ABB RAPID module: ABSACC.mod

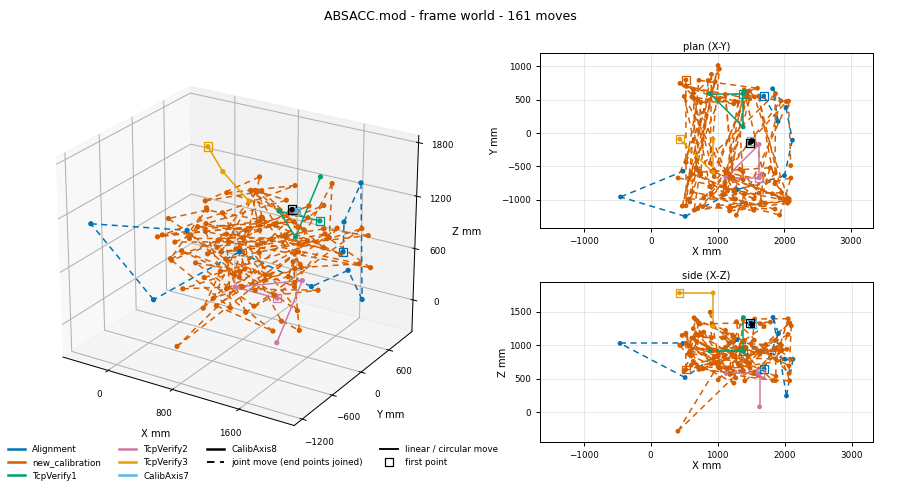
[picture p0: tool path of ABSACC.mod in frame world, 161 of 263 moves have a stored position in this frame; points joined in program order, loops and branches not executed]
%%%
  VERSION:1
  LANGUAGE:ENGLISH
%%%

MODULE ABSACC

    VAR robtarget current_pos   ;
    VAR string log_string;
    VAR iodev file_no;
    VAR num number;
    VAR string outnumber;
    VAR jointtarget jt_current;
    VAR robtarget rt_current;


    VAR num x_pos;
    VAR num y_pos;
    VAR num z_pos;
    VAR num q1_pos;
    VAR num q2_pos;
    VAR num q3_pos;
    VAR num q4_pos;


    VAR jointtarget jpos_after_move;
    VAR jointtarget currentjoints;
    VAR num rob_axis_1;                 ! ????1???
    VAR num rob_axis_2;                 ! ????2???
    VAR num rob_axis_3;                 ! ????3???
    VAR num rob_axis_4;                 ! ????4???
    VAR num rob_axis_5;                 ! ????5???
    VAR num rob_axis_6;                 ! ????6???


CONST robtarget Calib_1:=[[523.49,799.57,640.63],[0.427271,0.615474,0.485528,0.450495],[-1,-1,1,1],[0,9.0000E+09,9.0000E+09,0.000922768,0.0198127,0.000536354]];
CONST robtarget Calib_2:=[[526.56,-1091.2,1181.6],[0.427248,0.615504,0.485478,0.450359],[-1,-1,1,1],[0,9.0000E+09,9.0000E+09,0.000922768,0.020546,0.000486039]];
CONST robtarget Calib_3:=[[720.62,792.84,639.99],[0.427499,0.615430,0.485283,0.450683],[-1,-1,1,1],[0,9.0000E+09,9.0000E+09,0.000922768,0.020546,0.000486039]];
CONST robtarget Calib_4:=[[1598.1,672.95,554.69],[0.427422,0.615259,0.485561,0.450647],[-2,-2,1,1],[0,9.0000E+09,9.0000E+09,0.000922768,0.0181016,0.000506165]];
CONST robtarget Calib_5:=[[1022.6,515.85,667.24],[0.427491,0.615409,0.485531,0.450370],[-2,-2,1,1],[0,9.0000E+09,9.0000E+09,0.000922768,0.0181016,0.000506165]];
CONST robtarget Calib_6:=[[573.72,-670.12,994.4],[0.427363,0.615467,0.485428,0.450324],[-1,-2,2,1],[0,9.0000E+09,9.0000E+09,0.000770224,0.0198127,0.000536354]];
CONST robtarget Calib_7:=[[723.98,-576.9,1336.5],[0.427491,0.615540,0.485574,0.450598],[-2,-2,1,1],[0,9.0000E+09,9.0000E+09,0.000922768,0.0181016,0.000506165]];
CONST robtarget Calib_8:=[[582.16,-1033.6,910.76],[0.427404,0.615425,0.485431,0.450648],[-1,-2,2,1],[0,9.0000E+09,9.0000E+09,0.000770224,0.0198127,0.000536354]];
CONST robtarget Calib_9:=[[1006.3,1014.5,850.46],[0.427169,0.615279,0.485385,0.450491],[-1,-1,1,1],[0,9.0000E+09,9.0000E+09,0.000922768,0.0198127,0.000536354]];
CONST robtarget Calib_10:=[[566.63,-990.26,872.37],[0.427234,0.615354,0.485638,0.450740],[-1,-1,1,1],[0,9.0000E+09,9.0000E+09,0.000922768,0.0198127,0.000536354]];
CONST robtarget Calib_11:=[[1269.8,-989.4,513.75],[0.427266,0.615492,0.485274,0.450510],[-1,-1,1,1],[0,9.0000E+09,9.0000E+09,0.000922768,0.020546,0.000486039]];
CONST robtarget Calib_12:=[[1116.4,-816.34,1225.6],[0.427348,0.615327,0.485558,0.450713],[-2,-2,1,1],[0,9.0000E+09,9.0000E+09,0.000922768,0.0181016,0.000506165]];
CONST robtarget Calib_13:=[[1482.7,514.18,659.18],[0.427130,0.615463,0.485370,0.450503],[-1,-2,2,1],[0,9.0000E+09,9.0000E+09,0.000770224,0.0198127,0.000536354]];
CONST robtarget Calib_14:=[[531.86,699.88,1033.4],[0.427259,0.615357,0.485446,0.450699],[-1,-1,1,1],[0,9.0000E+09,9.0000E+09,0.000922768,0.020546,0.000486039]];
CONST robtarget Calib_15:=[[635.74,656.93,761.23],[0.427346,0.615523,0.485389,0.450649],[-1,-1,1,1],[0,9.0000E+09,9.0000E+09,0.000922768,0.020546,0.000486039]];
CONST robtarget Calib_16:=[[1241.2,439.93,437],[0.427180,0.615539,0.485346,0.450641],[-2,-2,1,1],[0,9.0000E+09,9.0000E+09,0.000922768,0.0181016,0.000506165]];
CONST robtarget Calib_17:=[[612.86,545.6,1108.6],[0.427352,0.615273,0.485557,0.450373],[-2,-2,1,1],[0,9.0000E+09,9.0000E+09,0.000922768,0.0181016,0.000506165]];
CONST robtarget Calib_18:=[[856.4,789.38,964.12],[0.427443,0.615400,0.485449,0.450538],[-1,-1,1,1],[0,9.0000E+09,9.0000E+09,0.000922768,0.0198127,0.000536354]];
CONST robtarget Calib_19:=[[746.48,-623.31,1183.2],[0.427151,0.615444,0.485503,0.450550],[-1,-1,1,1],[0,9.0000E+09,9.0000E+09,0.000922768,0.0198127,0.000536354]];
CONST robtarget Calib_20:=[[498.99,549.58,619.65],[0.427533,0.615524,0.485442,0.450402],[-1,-1,1,1],[0,9.0000E+09,9.0000E+09,0.000922768,0.0198127,0.000536354]];
CONST robtarget Calib_21:=[[1260.9,-903.01,847.24],[0.427221,0.615530,0.485537,0.450347],[-1,-1,1,1],[0,9.0000E+09,9.0000E+09,0.000922768,0.0198127,0.000536354]];
CONST robtarget Calib_22:=[[1115.2,580.02,967.53],[0.427294,0.615266,0.485509,0.450741],[-1,-2,2,1],[0,9.0000E+09,9.0000E+09,0.000770224,0.0198127,0.000536354]];
CONST robtarget Calib_23:=[[1222.6,-669.28,1154.2],[0.427349,0.615383,0.485339,0.450300],[-1,-1,1,1],[0,9.0000E+09,9.0000E+09,0.000922768,0.0198127,0.000536354]];
CONST robtarget Calib_24:=[[1384,-699.69,623.11],[0.427265,0.615494,0.485307,0.450350],[-1,-1,1,1],[0,9.0000E+09,9.0000E+09,0.000922768,0.020546,0.000486039]];
CONST robtarget Calib_25:=[[1308.7,467.72,716.41],[0.427497,0.615508,0.485570,0.450737],[-1,-2,2,1],[0,9.0000E+09,9.0000E+09,0.000770224,0.0198127,0.000536354]];
CONST robtarget Calib_26:=[[1108.9,-758.92,1117],[0.427089,0.615547,0.485259,0.450374],[-2,-2,1,1],[0,9.0000E+09,9.0000E+09,0.000922768,0.0181016,0.000506165]];
CONST robtarget Calib_27:=[[701,-1126.7,1157],[0.427424,0.615529,0.485327,0.450564],[-1,-2,2,1],[0,9.0000E+09,9.0000E+09,0.000770224,0.0198127,0.000536354]];
CONST robtarget Calib_28:=[[792.13,-971.51,1198.2],[0.427131,0.615367,0.485491,0.450773],[-2,-2,1,1],[0,9.0000E+09,9.0000E+09,0.000922768,0.0181016,0.000506165]];
CONST robtarget Calib_29:=[[1126,-591.56,665.82],[0.427307,0.615501,0.485324,0.450344],[-1,-1,1,1],[0,9.0000E+09,9.0000E+09,0.000922768,0.020546,0.000486039]];
CONST robtarget Calib_30:=[[635.98,600.07,1249.9],[0.427092,0.615395,0.485545,0.450727],[-1,-1,1,1],[0,9.0000E+09,9.0000E+09,0.000922768,0.0198127,0.000536354]];
CONST robtarget Calib_31:=[[674,-522.19,1382.2],[0.427363,0.615521,0.485308,0.450727],[-1,-2,2,1],[0,9.0000E+09,9.0000E+09,0.000770224,0.0198127,0.000536354]];
CONST robtarget Calib_32:=[[748.13,462.02,1157.5],[0.427338,0.615483,0.485637,0.450429],[-1,-2,2,1],[0,9.0000E+09,9.0000E+09,0.000770224,0.0198127,0.000536354]];
CONST robtarget Calib_33:=[[1259.1,477.91,827.2],[0.427346,0.615281,0.485321,0.450436],[-1,-2,2,1],[0,9.0000E+09,9.0000E+09,0.000770224,0.0198127,0.000536354]];
CONST robtarget Calib_34:=[[435.05,747.18,1000.2],[0.427446,0.615477,0.485492,0.450579],[-2,-2,1,1],[0,9.0000E+09,9.0000E+09,0.000922768,0.0181016,0.000506165]];
CONST robtarget Calib_35:=[[700.02,500.97,685.14],[0.427265,0.615499,0.485337,0.450378],[-1,-1,1,1],[0,9.0000E+09,9.0000E+09,0.000922768,0.0198127,0.000536354]];
CONST robtarget Calib_36:=[[527.77,-439.15,1030.3],[0.427281,0.615357,0.485288,0.450618],[-1,-1,1,1],[0,9.0000E+09,9.0000E+09,0.000922768,0.0198127,0.000536354]];
CONST robtarget Calib_37:=[[964.85,768.97,744],[0.427293,0.615355,0.485428,0.450593],[-2,-2,1,1],[0,9.0000E+09,9.0000E+09,0.000922768,0.0181016,0.000506165]];
CONST robtarget Calib_38:=[[469.94,-1095.9,1149],[0.427187,0.615553,0.485531,0.450739],[-1,-1,1,1],[0,9.0000E+09,9.0000E+09,0.000922768,0.0198127,0.000536354]];
CONST robtarget Calib_39:=[[908.06,882.12,1111.7],[0.427135,0.615427,0.485420,0.450717],[-2,-2,1,1],[0,9.0000E+09,9.0000E+09,0.000922768,0.0181016,0.000506165]];
CONST robtarget Calib_40:=[[889.34,-450.25,1494.7],[0.427395,0.615312,0.485584,0.450720],[-2,-2,1,1],[0,9.0000E+09,9.0000E+09,0.000922768,0.0181016,0.000506165]];
CONST robtarget Calib_41:=[[1026.6,961.76,736],[0.427363,0.615234,0.485457,0.450402],[-1,-1,1,1],[0,9.0000E+09,9.0000E+09,0.000922768,0.020546,0.000486039]];
CONST robtarget Calib_42:=[[406.52,-673.62,-280.36],[0.427280,0.615259,0.485296,0.450679],[-1,-1,1,1],[0,9.0000E+09,9.0000E+09,0.000922768,0.020546,0.000486039]];
CONST robtarget Calib_43:=[[2074.8,-1023.6,1336],[0.337031,0.670436,0.287182,0.595360],[-1,-1,1,1],[9.0000E+09,9.0000E+09,9.0000E+09,9.0000E+09,9.0000E+09,9.0000E+09]];
CONST robtarget Calib_44:=[[1181.5,-1112.6,566.66],[0.337038,0.670376,0.287151,0.595390],[-1,-1,2,1],[9.0000E+09,9.0000E+09,9.0000E+09,9.0000E+09,9.0000E+09,9.0000E+09]];
CONST robtarget Calib_45:=[[1861.9,-1141,473.33],[0.337097,0.670438,0.287154,0.595390],[-1,0,1,1],[9.0000E+09,9.0000E+09,9.0000E+09,9.0000E+09,9.0000E+09,9.0000E+09]];
CONST robtarget Calib_46:=[[901.25,-902.02,725.94],[0.337013,0.670422,0.287231,0.595328],[-1,-1,1,1],[9.0000E+09,9.0000E+09,9.0000E+09,9.0000E+09,9.0000E+09,9.0000E+09]];
CONST robtarget Calib_47:=[[1948.9,483.67,997.95],[0.337045,0.670418,0.287223,0.595385],[-1,-1,1,1],[9.0000E+09,9.0000E+09,9.0000E+09,9.0000E+09,9.0000E+09,9.0000E+09]];
CONST robtarget Calib_48:=[[1546.2,-986.65,603.41],[0.337073,0.670424,0.287150,0.595345],[0,0,1,1],[9.0000E+09,9.0000E+09,9.0000E+09,9.0000E+09,9.0000E+09,9.0000E+09]];
CONST robtarget Calib_49:=[[605.19,-604.49,704.07],[0.337059,0.670417,0.287152,0.595308],[0,0,1,1],[9.0000E+09,9.0000E+09,9.0000E+09,9.0000E+09,9.0000E+09,9.0000E+09]];
CONST robtarget Calib_50:=[[1718.7,-1051.7,1013.8],[0.337045,0.670449,0.287202,0.595417],[0,0,0,1],[9.0000E+09,9.0000E+09,9.0000E+09,9.0000E+09,9.0000E+09,9.0000E+09]];
CONST robtarget Calib_51:=[[1182.6,-676.82,1033.8],[0.337024,0.670403,0.287174,0.595407],[-1,-1,2,1],[9.0000E+09,9.0000E+09,9.0000E+09,9.0000E+09,9.0000E+09,9.0000E+09]];
CONST robtarget Calib_52:=[[1545.3,-1159,1076.6],[0.337084,0.670398,0.287161,0.595421],[0,0,1,1],[9.0000E+09,9.0000E+09,9.0000E+09,9.0000E+09,9.0000E+09,9.0000E+09]];
CONST robtarget Calib_53:=[[774.81,-1104.3,649.63],[0.337065,0.670394,0.287225,0.595345],[0,1,0,1],[9.0000E+09,9.0000E+09,9.0000E+09,9.0000E+09,9.0000E+09,9.0000E+09]];
CONST robtarget Calib_54:=[[1176.9,-617.93,582.71],[0.337054,0.670449,0.287235,0.595440],[0,0,0,1],[9.0000E+09,9.0000E+09,9.0000E+09,9.0000E+09,9.0000E+09,9.0000E+09]];
CONST robtarget Calib_55:=[[1933.5,-974.06,1016],[0.337054,0.670455,0.287213,0.595317],[-1,-1,1,1],[9.0000E+09,9.0000E+09,9.0000E+09,9.0000E+09,9.0000E+09,9.0000E+09]];
CONST robtarget Calib_56:=[[2052.5,-974.74,1397.5],[0.337096,0.670387,0.287178,0.595388],[0,0,1,1],[9.0000E+09,9.0000E+09,9.0000E+09,9.0000E+09,9.0000E+09,9.0000E+09]];
CONST robtarget Calib_57:=[[1552.8,542.67,1393.9],[0.337078,0.670388,0.287224,0.595338],[0,0,1,1],[9.0000E+09,9.0000E+09,9.0000E+09,9.0000E+09,9.0000E+09,9.0000E+09]];
CONST robtarget Calib_58:=[[1479.6,633.54,729.48],[0.337077,0.670453,0.287230,0.595399],[-1,-1,1,1],[9.0000E+09,9.0000E+09,9.0000E+09,9.0000E+09,9.0000E+09,9.0000E+09]];
CONST robtarget Calib_59:=[[942.08,-556.73,811.34],[0.337051,0.670394,0.287182,0.595426],[0,0,1,1],[9.0000E+09,9.0000E+09,9.0000E+09,9.0000E+09,9.0000E+09,9.0000E+09]];
CONST robtarget Calib_60:=[[1865.4,-737.13,799.35],[0.337079,0.670347,0.287195,0.595413],[0,0,1,1],[9.0000E+09,9.0000E+09,9.0000E+09,9.0000E+09,9.0000E+09,9.0000E+09]];
CONST robtarget Calib_61:=[[2050.6,-1051.8,1162.8],[0.337039,0.670451,0.287233,0.595373],[-1,-1,2,1],[9.0000E+09,9.0000E+09,9.0000E+09,9.0000E+09,9.0000E+09,9.0000E+09]];
CONST robtarget Calib_62:=[[1179.9,-1167.8,668.09],[0.337018,0.670357,0.287230,0.595352],[0,0,1,1],[9.0000E+09,9.0000E+09,9.0000E+09,9.0000E+09,9.0000E+09,9.0000E+09]];
CONST robtarget Calib_63:=[[1250.1,-852.23,1106.8],[0.337032,0.670393,0.287200,0.595412],[0,0,1,1],[9.0000E+09,9.0000E+09,9.0000E+09,9.0000E+09,9.0000E+09,9.0000E+09]];
CONST robtarget Calib_64:=[[1380.7,-581.78,1383.3],[0.337027,0.670421,0.287218,0.595331],[-2,-2,2,1],[9.0000E+09,9.0000E+09,9.0000E+09,9.0000E+09,9.0000E+09,9.0000E+09]];
CONST robtarget Calib_65:=[[1335.1,-543.79,968.31],[0.337051,0.670354,0.287205,0.595374],[0,1,0,1],[9.0000E+09,9.0000E+09,9.0000E+09,9.0000E+09,9.0000E+09,9.0000E+09]];
CONST robtarget Calib_66:=[[1622.8,-900.39,876.91],[0.337041,0.670454,0.287187,0.595438],[0,0,0,1],[9.0000E+09,9.0000E+09,9.0000E+09,9.0000E+09,9.0000E+09,9.0000E+09]];
CONST robtarget Calib_67:=[[1861.8,-601.93,954.03],[0.337062,0.670370,0.287184,0.595412],[-1,-1,2,1],[9.0000E+09,9.0000E+09,9.0000E+09,9.0000E+09,9.0000E+09,9.0000E+09]];
CONST robtarget Calib_68:=[[1869.1,592.3,538],[0.337015,0.670426,0.287199,0.595320],[0,0,1,1],[9.0000E+09,9.0000E+09,9.0000E+09,9.0000E+09,9.0000E+09,9.0000E+09]];
CONST robtarget Calib_69:=[[692.16,-548.27,1056.3],[0.337058,0.670360,0.287213,0.595396],[-2,-2,2,1],[9.0000E+09,9.0000E+09,9.0000E+09,9.0000E+09,9.0000E+09,9.0000E+09]];
CONST robtarget Calib_70:=[[1101.7,-909.92,848.42],[0.337048,0.670416,0.287158,0.595327],[-1,-1,2,1],[9.0000E+09,9.0000E+09,9.0000E+09,9.0000E+09,9.0000E+09,9.0000E+09]];
CONST robtarget Calib_71:=[[1007.8,-1088,485.37],[0.337071,0.670388,0.287186,0.595329],[0,1,0,1],[9.0000E+09,9.0000E+09,9.0000E+09,9.0000E+09,9.0000E+09,9.0000E+09]];
CONST robtarget Calib_72:=[[1421.7,-1049.4,969.62],[0.337024,0.670400,0.287209,0.595388],[-2,-2,2,1],[9.0000E+09,9.0000E+09,9.0000E+09,9.0000E+09,9.0000E+09,9.0000E+09]];
CONST robtarget Calib_73:=[[617.49,-882.09,948.54],[0.337019,0.670425,0.287148,0.595386],[-1,-1,1,1],[9.0000E+09,9.0000E+09,9.0000E+09,9.0000E+09,9.0000E+09,9.0000E+09]];
CONST robtarget Calib_74:=[[1931.9,-1230.9,917.13],[0.337103,0.670350,0.287183,0.595318],[0,1,0,1],[9.0000E+09,9.0000E+09,9.0000E+09,9.0000E+09,9.0000E+09,9.0000E+09]];
CONST robtarget Calib_75:=[[2100.7,-673.62,791.58],[0.337065,0.670443,0.287160,0.595345],[-1,0,1,1],[9.0000E+09,9.0000E+09,9.0000E+09,9.0000E+09,9.0000E+09,9.0000E+09]];
CONST robtarget Calib_76:=[[1149.7,-869.76,649.62],[0.337094,0.670428,0.287147,0.595325],[-1,0,1,1],[9.0000E+09,9.0000E+09,9.0000E+09,9.0000E+09,9.0000E+09,9.0000E+09]];
CONST robtarget Calib_77:=[[1431.9,625.97,764.27],[0.337014,0.670388,0.287161,0.595331],[-1,-1,2,1],[9.0000E+09,9.0000E+09,9.0000E+09,9.0000E+09,9.0000E+09,9.0000E+09]];
CONST robtarget Calib_78:=[[949.02,-653.32,926.53],[0.337059,0.670433,0.287179,0.595404],[-1,0,1,1],[9.0000E+09,9.0000E+09,9.0000E+09,9.0000E+09,9.0000E+09,9.0000E+09]];
CONST robtarget Calib_79:=[[640.82,524,1107.8],[0.337046,0.670413,0.287183,0.595344],[-1,-1,2,1],[9.0000E+09,9.0000E+09,9.0000E+09,9.0000E+09,9.0000E+09,9.0000E+09]];
CONST robtarget Calib_80:=[[881.01,-803.61,947.89],[0.337084,0.670403,0.287189,0.595343],[0,1,0,1],[9.0000E+09,9.0000E+09,9.0000E+09,9.0000E+09,9.0000E+09,9.0000E+09]];
CONST robtarget Calib_81:=[[2031.7,473.01,942.05],[0.337084,0.670381,0.287185,0.595336],[0,0,1,1],[9.0000E+09,9.0000E+09,9.0000E+09,9.0000E+09,9.0000E+09,9.0000E+09]];
CONST robtarget Calib_82:=[[1448.7,566.46,849.39],[0.337036,0.670409,0.287180,0.595326],[0,0,1,1],[9.0000E+09,9.0000E+09,9.0000E+09,9.0000E+09,9.0000E+09,9.0000E+09]];
CONST robtarget Calib_83:=[[1072.2,-924.1,1112.3],[0.337049,0.670411,0.287235,0.595327],[0,0,0,1],[9.0000E+09,9.0000E+09,9.0000E+09,9.0000E+09,9.0000E+09,9.0000E+09]];
CONST robtarget Calib_84:=[[1398.2,648.97,1074.8],[0.337050,0.670360,0.287199,0.595382],[-1,-1,1,1],[9.0000E+09,9.0000E+09,9.0000E+09,9.0000E+09,9.0000E+09,9.0000E+09]];
CONST robtarget Calib_85:=[[1692.1,-629.73,1280.4],[0.337086,0.670389,0.287196,0.595338],[-2,-2,2,1],[9.0000E+09,9.0000E+09,9.0000E+09,9.0000E+09,9.0000E+09,9.0000E+09]];
CONST robtarget Calib_86:=[[1635.2,-1070.1,1324.1],[0.337011,0.670430,0.287237,0.595376],[-1,-1,2,1],[9.0000E+09,9.0000E+09,9.0000E+09,9.0000E+09,9.0000E+09,9.0000E+09]];
CONST robtarget Calib_87:=[[1787,-520.57,1346.8],[0.337047,0.670444,0.287202,0.595388],[-1,-1,2,1],[9.0000E+09,9.0000E+09,9.0000E+09,9.0000E+09,9.0000E+09,9.0000E+09]];
CONST robtarget Calib_88:=[[735.47,-585.55,1318.4],[0.337086,0.670436,0.287148,0.595336],[-2,-2,2,1],[9.0000E+09,9.0000E+09,9.0000E+09,9.0000E+09,9.0000E+09,9.0000E+09]];
CONST robtarget Calib_89:=[[647.3,-1156,1412],[0.337021,0.670442,0.287213,0.595341],[-1,-1,2,1],[9.0000E+09,9.0000E+09,9.0000E+09,9.0000E+09,9.0000E+09,9.0000E+09]];
CONST robtarget Calib_90:=[[2064.3,-1013.5,695.66],[0.337032,0.670388,0.287233,0.595308],[0,0,0,1],[9.0000E+09,9.0000E+09,9.0000E+09,9.0000E+09,9.0000E+09,9.0000E+09]];
CONST robtarget Calib_91:=[[914.78,-574.42,1323.8],[0.337011,0.670425,0.287187,0.595439],[-1,-1,2,1],[9.0000E+09,9.0000E+09,9.0000E+09,9.0000E+09,9.0000E+09,9.0000E+09]];
CONST robtarget Calib_92:=[[1822.4,-911.38,476.82],[0.337067,0.670456,0.287225,0.595396],[-1,-1,1,1],[9.0000E+09,9.0000E+09,9.0000E+09,9.0000E+09,9.0000E+09,9.0000E+09]];
CONST robtarget Calib_93:=[[2074.2,-987.78,472.31],[0.337079,0.670363,0.287184,0.595396],[-1,-1,2,1],[9.0000E+09,9.0000E+09,9.0000E+09,9.0000E+09,9.0000E+09,9.0000E+09]];
CONST robtarget Calib_94:=[[1860.3,-759.59,1077.8],[0.337047,0.670419,0.287236,0.595422],[-2,-2,2,1],[9.0000E+09,9.0000E+09,9.0000E+09,9.0000E+09,9.0000E+09,9.0000E+09]];
CONST robtarget Calib_95:=[[1614.9,555.68,899.4],[0.337047,0.670434,0.287180,0.595372],[0,0,0,1],[9.0000E+09,9.0000E+09,9.0000E+09,9.0000E+09,9.0000E+09,9.0000E+09]];
CONST robtarget Calib_96:=[[1960.6,-894.35,930.39],[0.337070,0.670442,0.287225,0.595321],[-1,-1,2,1],[9.0000E+09,9.0000E+09,9.0000E+09,9.0000E+09,9.0000E+09,9.0000E+09]];
CONST robtarget Calib_97:=[[1405.1,-914.47,469.92],[0.337108,0.670454,0.287208,0.595360],[0,1,0,1],[9.0000E+09,9.0000E+09,9.0000E+09,9.0000E+09,9.0000E+09,9.0000E+09]];
CONST robtarget Calib_98:=[[1281,-1232.4,1353.2],[0.337026,0.670376,0.287182,0.595400],[-2,-2,2,1],[9.0000E+09,9.0000E+09,9.0000E+09,9.0000E+09,9.0000E+09,9.0000E+09]];
CONST robtarget Calib_99:=[[2064.8,479.5,583.13],[0.337055,0.670394,0.287212,0.595368],[0,0,1,1],[9.0000E+09,9.0000E+09,9.0000E+09,9.0000E+09,9.0000E+09,9.0000E+09]];
CONST robtarget Calib_100:=[[2097.5,-487.03,1291.9],[0.337063,0.670458,0.287190,0.595322],[-1,-1,2,1],[9.0000E+09,9.0000E+09,9.0000E+09,9.0000E+09,9.0000E+09,9.0000E+09]];







CONST jointtarget JT_Set1_1:=[[53.1735,26.9510,23.3573,73.4890,-59.9300,59.2650],[0,9000000000.0,9000000000.0,0,0,0]];
CONST jointtarget JT_Set1_2:=[[104.8875,-39.2172,32.0501,101.4420,-111.1420,5.5760],[0,9000000000.0,9000000000.0,0,0,0]];
CONST jointtarget JT_Set1_3:=[[-0.5260,-0.9171,-22.1124,172.3270,-36.5000,-74.4910],[0,9000000000.0,9000000000.0,0,0,0]];
CONST jointtarget JT_Set1_4:=[[-71.4352,25.7651,25.2310,-79.7280,-64.8550,137.7380],[0,9000000000.0,9000000000.0,0,0,0]];
CONST jointtarget JT_Set1_5:=[[-33.2693,73.5127,6.3150,-29.5740,-67.8700,103.3770],[0,9000000000.0,9000000000.0,0,0,0]];
CONST jointtarget JT_Set1_6:=[[-10.4906,14.7639,-6.2399,-133.2560,-7.0380,230.5130],[0,9000000000.0,9000000000.0,0,0,0]];
CONST jointtarget JT_Set1_7:=[[-93.3527,9.8440,13.8280,-101.4370,-83.0510,165.4770],[0,9000000000.0,9000000000.0,0,0,0]];
CONST jointtarget JT_Set1_8:=[[11.7457,37.5557,36.3356,18.9030,-61.4260,92.9380],[0,9000000000.0,9000000000.0,0,0,0]];
CONST jointtarget JT_Set1_9:=[[21.7410,14.7129,-20.7875,125.9430,-33.0750,-25.9510],[0,9000000000.0,9000000000.0,0,0,0]];
CONST jointtarget JT_Set1_10:=[[-2.9191,4.9374,-1.3727,167.2410,-9.9250,-68.6510],[0,9000000000.0,9000000000.0,0,0,0]];
CONST jointtarget JT_Set1_11:=[[-5.6872,43.8374,27.8881,-61.6498,-69.5127,61.2],[0,9000000000.0,9000000000.0,0,0,0]];
CONST jointtarget JT_Set1_12:=[[50.3079,41.8227,-20.4018,120.7182,-152.8732,-46.8],[0,9000000000.0,9000000000.0,0,0,0]];
CONST jointtarget JT_Set1_13:=[[84.3385,18.9432,34.5532,160.8424,-29.5414,-118.8],[0,9000000000.0,9000000000.0,0,0,0]];
CONST jointtarget JT_Set1_14:=[[58.297,-2.0746,27.5285,-154.2974,-61.9657,-72.0],[0,9000000000.0,9000000000.0,0,0,0]];
CONST jointtarget JT_Set1_15:=[[32.8735,-30.4364,-59.6442,95.92,-47.9329,-86.4],[0,9000000000.0,9000000000.0,0,0,0]];
CONST jointtarget JT_Set1_16:=[[-33.6427,-18.5643,-12.0604,48.1328,-64.5324,126.0],[0,9000000000.0,9000000000.0,0,0,0]];
CONST jointtarget JT_Set1_17:=[[70.3802,17.2132,-4.0173,-21.5256,-130.5416,43.2],[0,9000000000.0,9000000000.0,0,0,0]];
CONST jointtarget JT_Set1_18:=[[89.0267,-51.2569,56.4018,-36.8517,-171.8904,-39.6],[0,9000000000.0,9000000000.0,0,0,0]];
CONST jointtarget JT_Set1_19:=[[5.7192,-2.5391,54.5482,-94.111,-150.4586,75.6],[0,9000000000.0,9000000000.0,0,0,0]];
CONST jointtarget JT_Set1_20:=[[-0.2027,50.2882,-24.7763,71.1219,-88.2809,97.2],[0,9000000000.0,9000000000.0,0,0,0]];
CONST jointtarget JT_Set1_21:=[[40.4823,-51.699,50.7331,136.0443,-70.7312,162.0],[0,9000000000.0,9000000000.0,0,0,0]];
CONST jointtarget JT_Set1_22:=[[-80.423,25.9753,1.6904,-171.4325,-135.2349,-75.6],[0,9000000000.0,9000000000.0,0,0,0]];
CONST jointtarget JT_Set1_23:=[[11.1889,-11.9535,-14.0107,-141.8983,-94.014,108.0],[0,9000000000.0,9000000000.0,0,0,0]];
CONST jointtarget JT_Set1_24:=[[54.1566,23.8297,-25.9466,8.0085,-89.427,165.6],[0,9000000000.0,9000000000.0,0,0,0]];
CONST jointtarget JT_Set1_25:=[[-59.19,39.8806,42.4357,-114.1731,-100.9528,-97.2],[0,9000000000.0,9000000000.0,0,0,0]];
CONST jointtarget JT_Set1_26:=[[22.8731,-54.4881,33.5123,-146.6343,-111.7156,-28.8],[0,9000000000.0,9000000000.0,0,0,0]];
CONST jointtarget JT_Set1_27:=[[-17.9117,51.6859,-47.3684,-76.9759,-37.8145,-50.4],[0,9000000000.0,9000000000.0,0,0,0]];
CONST jointtarget JT_Set1_28:=[[66.8969,-54.1454,-30.6363,156.1064,-124.7502,7.2],[0,9000000000.0,9000000000.0,0,0,0]];
CONST jointtarget JT_Set1_29:=[[27.4745,30.9191,-59.737,55.7958,-158.4348,28.8],[0,9000000000.0,9000000000.0,0,0,0]];
CONST jointtarget JT_Set1_30:=[[-14.9131,37.7906,30.1398,75.8579,-55.2498,21.6],[0,9000000000.0,9000000000.0,0,0,0]];
CONST jointtarget JT_Set1_31:=[[3.0179,52.3778,-47.9993,-78.7849,-44.7651,-140.4],[0,9000000000.0,9000000000.0,0,0,0]];
CONST jointtarget JT_Set1_32:=[[-83.9819,-55.1498,-7.8347,108.3191,-115.4676,79.2],[0,9000000000.0,9000000000.0,0,0,0]];
CONST jointtarget JT_Set1_33:=[[25.0821,42.0558,5.111,-1.4635,-85.986,-115.2],[0,9000000000.0,9000000000.0,0,0,0]];
CONST jointtarget JT_Set1_34:=[[76.0705,-26.6255,7.5352,30.9977,-14.0699,-111.6],[0,9000000000.0,9000000000.0,0,0,0]];
CONST jointtarget JT_Set1_35:=[[19.3661,-58.9602,39.5929,-86.448,-116.7437,-10.8],[0,9000000000.0,9000000000.0,0,0,0]];
CONST jointtarget JT_Set1_36:=[[80.2267,36.5199,-43.3022,143.7073,-46.3699,57.6],[0,9000000000.0,9000000000.0,0,0,0]];
CONST jointtarget JT_Set1_37:=[[48.0395,-22.389,-23.9848,-24.4526,-136.8864,-68.4],[0,9000000000.0,9000000000.0,0,0,0]];
CONST jointtarget JT_Set1_38:=[[18.7521,-39.7648,-9.1071,80.5939,-43.1136,-169.2],[0,9000000000.0,9000000000.0,0,0,0]];
CONST jointtarget JT_Set1_39:=[[-19.8231,-9.8027,-49.6534,92.993,-118.0343,82.8],[0,9000000000.0,9000000000.0,0,0,0]];
CONST jointtarget JT_Set1_40:=[[-74.0487,-29.5339,-27.7307,15.6716,-91.7191,-180.0],[0,9000000000.0,9000000000.0,0,0,0]];
CONST jointtarget JT_Set1_41:=[[66.8104,2.6569,-16.8701,-179.0955,-35.9041,158.4],[0,9000000000.0,9000000000.0,0,0,0]];
CONST jointtarget JT_Set1_42:=[[-86.0097,10.1224,-50.2238,-46.3238,-90.573,-61.2],[0,9000000000.0,9000000000.0,0,0,0]];
CONST jointtarget JT_Set1_43:=[[65.7842,-4.3144,-8.6083,68.1949,-142.1855,64.8],[0,9000000000.0,9000000000.0,0,0,0]];
CONST jointtarget JT_Set1_44:=[[-79.6292,30.4972,51.7061,128.3812,-109.2688,122.4],[0,9000000000.0,9000000000.0,0,0,0]];
CONST jointtarget JT_Set1_45:=[[17.1694,43.2389,9.1874,-101.7741,-63.2563,-90.0],[0,9000000000.0,9000000000.0,0,0,0]];
CONST jointtarget JT_Set1_46:=[[-56.1143,39.1682,27.6415,-66.3859,-57.9945,36.0],[0,9000000000.0,9000000000.0,0,0,0]];
CONST jointtarget JT_Set1_47:=[[-0.1178,8.7955,47.1428,115.9821,-104.4775,0.0],[0,9000000000.0,9000000000.0,0,0,0]];
CONST jointtarget JT_Set1_48:=[[-0.9982,-4.9911,-14.7009,35.7337,-56.633,86.4],[0,9000000000.0,9000000000.0,0,0,0]];
CONST jointtarget JT_Set1_49:=[[43.6689,41.9657,25.2907,-109.4371,-76.7029,-108.0],[0,9000000000.0,9000000000.0,0,0,0]];
CONST jointtarget JT_Set1_50:=[[18.1302,-40.4613,16.8971,-134.2353,-80.2122,-82.8],[0,9000000000.0,9000000000.0,0,0,0]];
CONST jointtarget JT_Set1_51:=[[-9.9137,59.6392,-58.603,38.6607,-99.7878,-57.6],[0,9000000000.0,9000000000.0,0,0,0]];
CONST jointtarget JT_Set1_52:=[[65.4327,3.1725,49.9096,-49.2508,-31.7883,-14.4],[0,9000000000.0,9000000000.0,0,0,0]];
CONST jointtarget JT_Set1_53:=[[60.6536,14.2971,40.2438,-126.5722,-105.6643,-136.8],[0,9000000000.0,9000000000.0,0,0,0]];
CONST jointtarget JT_Set1_54:=[[68.6718,-24.5563,46.7768,51.0598,-98.6269,10.8],[0,9000000000.0,9000000000.0,0,0,0]];
CONST jointtarget JT_Set1_55:=[[14.1083,-57.6796,40.3064,91.184,-81.3731,32.4],[0,9000000000.0,9000000000.0,0,0,0]];
CONST jointtarget JT_Set1_56:=[[-23.3421,18.6099,-2.3236,-13.8626,-119.3406,118.8],[0,9000000000.0,9000000000.0,0,0,0]];
CONST jointtarget JT_Set1_57:=[[-78.128,-10.492,19.6883,-129.4992,-68.2844,129.6],[0,9000000000.0,9000000000.0,0,0,0]];
CONST jointtarget JT_Set1_58:=[[-35.7881,25.0118,35.0866,-159.0334,-114.2048,-172.8],[0,9000000000.0,9000000000.0,0,0,0]];
CONST jointtarget JT_Set1_59:=[[65.3047,-8.5084,47.4423,-53.9868,-84.8364,-154.8],[0,9000000000.0,9000000000.0,0,0,0]];
CONST jointtarget JT_Set1_60:=[[56.0198,56.5793,-5.1291,-41.5877,-97.4696,46.8],[0,9000000000.0,9000000000.0,0,0,0]];
CONST jointtarget JT_Set1_61:=[[59.2313,14.8881,-51.7701,-161.9604,-50.9499,-36.0],[0,9000000000.0,9000000000.0,0,0,0]];
CONST jointtarget JT_Set1_62:=[[47.4907,-56.6752,-59.2606,111.2461,-138.5904,154.8],[0,9000000000.0,9000000000.0,0,0,0]];
CONST jointtarget JT_Set1_63:=[[86.8852,29.0221,11.4042,43.3967,-102.1224,169.2],[0,9000000000.0,9000000000.0,0,0,0]];
CONST jointtarget JT_Set1_64:=[[-22.2175,-45.0242,33.717,-69.3129,-67.0455,140.4],[0,9000000000.0,9000000000.0,0,0,0]];
CONST jointtarget JT_Set1_65:=[[-30.5017,12.5155,58.7496,-131.3082,-120.6638,100.8],[0,9000000000.0,9000000000.0,0,0,0]];
CONST jointtarget JT_Set1_66:=[[-6.0579,-38.7443,27.8748,153.1793,-21.5652,50.4],[0,9000000000.0,9000000000.0,0,0,0]];
CONST jointtarget JT_Set1_67:=[[-87.1488,-45.1791,29.9886,113.0551,-24.4946,-25.2],[0,9000000000.0,9000000000.0,0,0,0]];
CONST jointtarget JT_Set1_68:=[[-54.6928,-49.7576,48.3583,123.6452,-165.9301,-79.2],[0,9000000000.0,9000000000.0,0,0,0]];
CONST jointtarget JT_Set1_69:=[[32.4759,54.5816,-50.9787,145.5163,-140.3539,176.4],[0,9000000000.0,9000000000.0,0,0,0]];
CONST jointtarget JT_Set1_70:=[[-21.1681,-53.3341,35.2605,83.521,-33.9013,-176.4],[0,9000000000.0,9000000000.0,0,0,0]];
CONST jointtarget JT_Set1_71:=[[71.0062,59.2081,23.1351,-9.1266,-73.142,144.0],[0,9000000000.0,9000000000.0,0,0,0]];
CONST jointtarget JT_Set1_72:=[[-46.8827,49.7226,19.3473,3.2725,-74.3357,-126.0],[0,9000000000.0,9000000000.0,0,0,0]];
CONST jointtarget JT_Set1_73:=[[33.0473,-0.4275,-32.8505,165.5784,-110.4873,25.2],[0,9000000000.0,9000000000.0,0,0,0]];
CONST jointtarget JT_Set1_74:=[[-3.3169,-55.5535,-40.2605,-163.7694,-144.0959,172.8],[0,9000000000.0,9000000000.0,0,0,0]];
CONST jointtarget JT_Set1_75:=[[38.5615,10.8124,53.7453,-81.712,-133.6301,-100.8],[0,9000000000.0,9000000000.0,0,0,0]];
CONST jointtarget JT_Set1_76:=[[-66.2109,0.9579,51.2879,168.5054,-161.8051,136.8],[0,9000000000.0,9000000000.0,0,0,0]];
CONST jointtarget JT_Set1_77:=[[74.2661,-23.2977,-22.9478,103.5831,-41.4096,68.4],[0,9000000000.0,9000000000.0,0,0,0]];
CONST jointtarget JT_Set1_78:=[[-54.2679,-11.4899,-36.2264,-4.3905,-82.5304,-7.2],[0,9000000000.0,9000000000.0,0,0,0]];
CONST jointtarget JT_Set1_79:=[[-64.7589,36.4248,13.275,58.7228,-75.5225,-64.8],[0,9000000000.0,9000000000.0,0,0,0]];
CONST jointtarget JT_Set1_80:=[[49.3794,-17.4967,-35.3362,-26.2616,-27.1268,-104.4],[0,9000000000.0,9000000000.0,0,0,0]];
CONST jointtarget JT_Set1_81:=[[73.9919,-53.9951,58.2495,-98.8471,-96.3153,-147.6],[0,9000000000.0,9000000000.0,0,0,0]];
CONST jointtarget JT_Set1_82:=[[-30.5839,-56.1184,58.8879,-33.9247,-39.6461,-165.6],[0,9000000000.0,9000000000.0,0,0,0]];
CONST jointtarget JT_Set1_83:=[[13.8473,51.0523,-38.8346,176.1685,-65.7952,93.6],[0,9000000000.0,9000000000.0,0,0,0]];
CONST jointtarget JT_Set1_84:=[[29.3861,-31.423,-37.0438,63.4588,-59.3362,-129.6],[0,9000000000.0,9000000000.0,0,0,0]];
CONST jointtarget JT_Set1_85:=[[34.252,18.7358,-16.464,23.3346,-18.1949,-93.6],[0,9000000000.0,9000000000.0,0,0,0]];
CONST jointtarget JT_Set1_86:=[[9.4172,12.7556,-31.3028,148.4433,-92.866,-144.0],[0,9000000000.0,9000000000.0,0,0,0]];
CONST jointtarget JT_Set1_87:=[[6.08,45.5454,-3.9299,-16.7896,-148.2117,-133.2],[0,9000000000.0,9000000000.0,0,0,0]];
CONST jointtarget JT_Set1_88:=[[22.6408,-5.2826,-57.3996,60.5318,-49.4584,133.2],[0,9000000000.0,9000000000.0,0,0,0]];
CONST jointtarget JT_Set1_89:=[[22.0157,-20.4801,23.4061,-151.3703,-103.2971,54.0],[0,9000000000.0,9000000000.0,0,0,0]];
CONST jointtarget JT_Set1_90:=[[-14.8025,11.8095,-8.4351,-29.1887,-79.0472,-151.2],[0,9000000000.0,9000000000.0,0,0,0]];
CONST jointtarget JT_Set1_91:=[[-83.0002,41.4388,-15.5128,6.1995,-155.5054,151.2],[0,9000000000.0,9000000000.0,0,0,0]];
CONST jointtarget JT_Set1_92:=[[-3.1983,9.7239,39.5441,173.2415,-112.9545,90.0],[0,9000000000.0,9000000000.0,0,0,0]];
CONST jointtarget JT_Set1_93:=[[76.8431,12.8642,-26.0615,28.0706,-8.1096,-32.4],[0,9000000000.0,9000000000.0,0,0,0]];
CONST jointtarget JT_Set1_94:=[[-75.8227,28.4404,36.1849,140.7803,-83.6847,14.4],[0,9000000000.0,9000000000.0,0,0,0]];
CONST jointtarget JT_Set1_95:=[[-13.1952,-51.2187,-57.7856,88.257,-126.157,-18.0],[0,9000000000.0,9000000000.0,0,0,0]];
CONST jointtarget JT_Set1_96:=[[-30.8058,4.128,-20.2128,-74.0489,-123.367,104.4],[0,9000000000.0,9000000000.0,0,0,0]];
CONST jointtarget JT_Set1_97:=[[-47.0501,-48.2183,-39.1149,18.5986,-71.9408,147.6],[0,9000000000.0,9000000000.0,0,0,0]];
CONST jointtarget JT_Set1_98:=[[-34.4198,56.3357,-2.9773,-56.9138,-95.1636,-162.0],[0,9000000000.0,9000000000.0,0,0,0]];
CONST jointtarget JT_Set1_99:=[[-25.5576,-31.4078,37.83,-121.8362,-129.0501,-21.6],[0,9000000000.0,9000000000.0,0,0,0]];
CONST jointtarget JT_Set1_100:=[[-68.6709,-57.1729,-14.2882,133.1172,-53.843,39.6],[0,9000000000.0,9000000000.0,0,0,0]];


    PERS tooldata tool_abs:=[TRUE,[[58.5955,-73.8474,157.464],[1,0,0,0]],[4.7,[-65.7,-43.2,147.5],[1,0,0,0],0.122,0,0.009]];




    CONST robtarget Align_1:=[[1692.44,556.50,645.46],[0.33701,0.670346,0.287238,0.595445],[0,0,1,1],[9E+9,9E+9,9E+9,9E+9,9E+9,9E+9]];
    CONST robtarget Align_2:=[[1907.75,175.07,1175.48],[0.33701,0.670346,0.287238,0.595445],[0,0,0,1],[9E+9,9E+9,9E+9,9E+9,9E+9,9E+9]];
    CONST robtarget Align_3:=[[1825.50,665.72,1417.59],[0.33701,0.670346,0.287238,0.595445],[0,1,0,1],[9E+9,9E+9,9E+9,9E+9,9E+9,9E+9]];
    CONST robtarget Align_4:=[[2026.63,383.98,246.89],[0.337011,0.670346,0.287238,0.595444],[0,0,1,1],[9E+9,9E+9,9E+9,9E+9,9E+9,9E+9]];
    CONST robtarget Align_5:=[[2122.83,-105.59,794.02],[0.337011,0.670346,0.287238,0.595444],[-1,0,1,1],[9E+9,9E+9,9E+9,9E+9,9E+9,9E+9]];
    CONST robtarget Align_6:=[[2003.35,-638.19,793.93],[0.337039,0.670427,0.287216,0.595348],[-1,-1,1,1],[9E+9,9E+9,9E+9,9E+9,9E+9,9E+9]];
    CONST robtarget Align_7:=[[1289.99,-848.78,1084.42],[0.337112,0.670461,0.287143,0.595304],[-1,-1,2,1],[9E+9,9E+9,9E+9,9E+9,9E+9,9E+9]];
    CONST robtarget Align_8:=[[514.04,-1249.56,520.38],[0.337111,0.670461,0.287144,0.595304],[-1,-1,1,1],[9E+9,9E+9,9E+9,9E+9,9E+9,9E+9]];
    CONST robtarget Align_9:=[[-456.25,-958.05,1029.38],[0.337112,0.670461,0.287143,0.595304],[-2,-2,2,1],[9E+9,9E+9,9E+9,9E+9,9E+9,9E+9]];
    CONST robtarget Align_10:=[[481.95,-572.24,1029.38],[0.337112,0.670461,0.287143,0.595304],[-1,-1,2,1],[9E+9,9E+9,9E+9,9E+9,9E+9,9E+9]];


    CONST robtarget CalibAxis7_1:=[[1507.65,-121.92,1315.22],[0.63677,0.23804,0.733373,-0.00502791],[0,-2,1,0],[-0.00191984,-0.00315776,9E+09,9E+09,9E+09,9E+09]];
    CONST robtarget CalibAxis7_2:=[[1507.68,-121.92,1315.34],[0.636801,0.23803,0.733349,-0.00502536],[0,-2,1,0],[-8.81484,-0.00328435,9E+09,9E+09,9E+09,9E+09]];
    CONST robtarget CalibAxis7_3:=[[1507.68,-121.93,1315.34],[0.636801,0.238032,0.733348,-0.00502462],[0,-2,1,0],[-11.8361,-0.00315776,9E+09,9E+09,9E+09,9E+09]];
    CONST robtarget CalibAxis7_4:=[[1507.68,-121.93,1315.34],[0.636802,0.238029,0.733348,-0.00502757],[0,-2,1,0],[-15.9282,-0.00328435,9E+09,9E+09,9E+09,9E+09]];
    CONST robtarget CalibAxis7_5:=[[1507.68,-121.93,1315.34],[0.636802,0.238031,0.733348,-0.00502651],[0,-2,1,0],[-21.2393,-0.00138547,9E+09,9E+09,9E+09,9E+09]];
    CONST robtarget CalibAxis7_6:=[[1507.68,-121.93,1315.34],[0.636802,0.238031,0.733348,-0.00502574],[0,-2,1,0],[-25.5017,-0.0025248,9E+09,9E+09,9E+09,9E+09]];
    CONST robtarget CalibAxis7_7:=[[1507.68,-121.93,1315.34],[0.636801,0.238032,0.733349,-0.00502496],[0,-2,1,0],[-32.081,-0.0025248,9E+09,9E+09,9E+09,9E+09]];
    CONST robtarget CalibAxis7_8:=[[1507.68,-121.93,1315.34],[0.636802,0.238031,0.733348,-0.00502574],[0,-2,1,0],[-35.336,-0.0025248,9E+09,9E+09,9E+09,9E+09]];
    CONST robtarget CalibAxis7_9:=[[1507.68,-121.93,1315.34],[0.636802,0.238031,0.733348,-0.00502626],[0,-2,1,0],[-42.6204,-0.0025248,9E+09,9E+09,9E+09,9E+09]];
    CONST robtarget CalibAxis7_10:=[[1507.68,-121.92,1315.34],[0.636801,0.23803,0.733349,-0.00502622],[0,-2,1,0],[-51.3046,-0.00244041,9E+09,9E+09,9E+09,9E+09]];
    CONST robtarget CalibAxis7_11:=[[1507.68,-121.92,1315.34],[0.636802,0.238032,0.733348,-0.00502646],[0,-2,1,0],[-53.5742,-0.0025248,9E+09,9E+09,9E+09,9E+09]];
    CONST robtarget CalibAxis7_12:=[[1507.68,-121.92,1315.34],[0.636802,0.238031,0.733348,-0.00502491],[0,-2,1,0],[-56.2912,-0.0025248,9E+09,9E+09,9E+09,9E+09]];
    CONST robtarget CalibAxis7_13:=[[1507.68,-121.93,1315.34],[0.636802,0.238032,0.733348,-0.0050253],[0,-2,1,0],[-65.1938,-0.0025248,9E+09,9E+09,9E+09,9E+09]];
    CONST robtarget CalibAxis7_14:=[[1507.68,-121.93,1315.34],[0.636802,0.238032,0.733348,-0.0050253],[0,-2,1,0],[-72.2042,-0.0025248,9E+09,9E+09,9E+09,9E+09]];
    CONST robtarget CalibAxis7_15:=[[1507.68,-121.92,1315.34],[0.636802,0.23803,0.733348,-0.00502588],[0,-2,1,0],[-76.3963,-0.00244041,9E+09,9E+09,9E+09,9E+09]];
    CONST robtarget CalibAxis7_16:=[[1507.68,-121.92,1315.34],[0.636802,0.238031,0.733348,-0.00502414],[0,-2,1,0],[-81.4035,-0.00265139,9E+09,9E+09,9E+09,9E+09]];
    CONST robtarget CalibAxis7_17:=[[1507.68,-121.93,1315.34],[0.636801,0.238032,0.733348,-0.0050248],[0,-2,1,0],[-83.6198,-0.00244041,9E+09,9E+09,9E+09,9E+09]];
    CONST robtarget CalibAxis7_18:=[[1507.68,-121.93,1315.34],[0.636801,0.238032,0.733348,-0.00502462],[0,-2,1,0],[-88.5747,0.000597801,9E+09,9E+09,9E+09,9E+09]];
    CONST robtarget CalibAxis7_19:=[[1507.68,-121.93,1315.34],[0.636802,0.238032,0.733348,-0.00502545],[0,-2,1,0],[-89.3598,0.000682195,9E+09,9E+09,9E+09,9E+09]];
    CONST robtarget CalibAxis7_20:=[[1507.68,-121.93,1315.34],[0.636802,0.238029,0.733348,-0.00502757],[0,-2,1,0],[-89.996,0.000682195,9E+09,9E+09,9E+09,9E+09]];


	CONST robtarget CalibAxis8_1:=[[1480.22,-148.61,1332.38],[0.6547,0.27295,0.702593,-0.056821],[0,-2,1,0],[0.00442388,-0.00180745,9E+09,9E+09,9E+09,9E+09]];
    CONST robtarget CalibAxis8_2:=[[1480.21,-148.61,1332.32],[0.654685,0.272947,0.702608,-0.0568259],[0,-2,1,0],[0.00457674,2.86415,9E+09,9E+09,9E+09,9E+09]];
    CONST robtarget CalibAxis8_3:=[[1507.58,-121.94,1314.95],[0.636707,0.238034,0.733429,-0.00505452],[0,-2,1,0],[-0.00249306,15.3797,9E+09,9E+09,9E+09,9E+09]];
    CONST robtarget CalibAxis8_4:=[[1507.58,-121.94,1314.91],[0.636696,0.238033,0.733439,-0.00505943],[0,-2,1,0],[-0.00228288,17.8713,9E+09,9E+09,9E+09,9E+09]];
    CONST robtarget CalibAxis8_5:=[[1507.66,-121.93,1315.23],[0.636773,0.238027,0.733374,-0.00503567],[0,-2,1,0],[-0.002837,34.8691,9E+09,9E+09,9E+09,9E+09]];
    CONST robtarget CalibAxis8_6:=[[1507.66,-121.93,1315.22],[0.636773,0.238029,0.733374,-0.00503471],[0,-2,1,0],[-0.002837,52.666,9E+09,9E+09,9E+09,9E+09]];
    CONST robtarget CalibAxis8_7:=[[1507.66,-121.93,1315.23],[0.636773,0.238027,0.733374,-0.00503567],[0,-2,1,0],[-0.002837,89.6947,9E+09,9E+09,9E+09,9E+09]];
    CONST robtarget CalibAxis8_8:=[[1507.66,-121.93,1315.22],[0.636773,0.238029,0.733374,-0.00503471],[0,-2,1,0],[-0.002837,101.138,9E+09,9E+09,9E+09,9E+09]];
    CONST robtarget CalibAxis8_9:=[[1507.65,-121.93,1315.17],[0.636758,0.238026,0.733387,-0.00504157],[0,-2,1,0],[-0.00276057,137.405,9E+09,9E+09,9E+09,9E+09]];
    CONST robtarget CalibAxis8_10:=[[1507.64,-121.93,1315.11],[0.636744,0.238026,0.733399,-0.0050481],[0,-2,1,0],[-0.00251217,165.75,9E+09,9E+09,9E+09,9E+09]];
    CONST robtarget CalibAxis8_11:=[[1507.62,-121.93,1315.05],[0.636729,0.238027,0.733413,-0.00505148],[0,-2,1,0],[-0.00249306,200.212,9E+09,9E+09,9E+09,9E+09]];
    CONST robtarget CalibAxis8_12:=[[1507.60,-121.94,1314.93],[0.6367,0.238025,0.733438,-0.00506073],[0,-2,1,0],[-0.00241663,254.25,9E+09,9E+09,9E+09,9E+09]];
    CONST robtarget CalibAxis8_13:=[[1507.59,-121.94,1314.87],[0.636683,0.238025,0.733453,-0.00506355],[0,-2,1,0],[-0.00245485,295.246,9E+09,9E+09,9E+09,9E+09]];
    CONST robtarget CalibAxis8_14:=[[1507.58,-121.94,1314.81],[0.63667,0.238023,0.733465,-0.00507103],[0,-2,1,0],[-0.00251217,315.066,9E+09,9E+09,9E+09,9E+09]];
    CONST robtarget CalibAxis8_15:=[[1507.57,-121.93,1314.75],[0.636653,0.238022,0.73348,-0.00506991],[0,-2,1,0],[-0.00245485,326.236,9E+09,9E+09,9E+09,9E+09]];
    CONST robtarget CalibAxis8_16:=[[1507.56,-121.94,1314.69],[0.636639,0.238021,0.733492,-0.00507623],[0,-2,1,0],[-0.00241663,334.064,9E+09,9E+09,9E+09,9E+09]];
    CONST robtarget CalibAxis8_17:=[[1507.54,-121.94,1314.64],[0.636626,0.238016,0.733506,-0.00508646],[0,-2,1,0],[-0.00239753,348.831,9E+09,9E+09,9E+09,9E+09]];
    CONST robtarget CalibAxis8_18:=[[1507.52,-121.94,1314.52],[0.636597,0.23801,0.733532,-0.00509305],[0,-2,1,0],[-0.00211091,354.301,9E+09,9E+09,9E+09,9E+09]];
    CONST robtarget CalibAxis8_19:=[[1507.50,-121.93,1314.41],[0.636567,0.238005,0.73356,-0.00510047],[0,-2,1,0],[-0.00170965,358.199,9E+09,9E+09,9E+09,9E+09]];
    CONST robtarget CalibAxis8_20:=[[1507.49,-121.94,1314.35],[0.636554,0.238003,0.733572,-0.0051093],[0,-2,1,0],[-0.00163322,360,9E+09,9E+09,9E+09,9E+09]];
    TASK PERS wobjdata wobjabs:=[FALSE,TRUE,"",[[245.011,286.912,1531.74],[0.000293811,-0.000374324,-1,1.0986E-7]],[[0,0,0],[1,0,0,0]]];


  PROC Alignment()
    number :=1;
    MoveJ Align_1,v200,fine,tool_abs\WObj:=wobj0;
    err_write_jogposition;
    MoveJ Align_2,v200,fine,tool_abs\WObj:=wobj0;
    err_write_jogposition;
    MoveJ Align_3,v200,fine,tool_abs\WObj:=wobj0;
    err_write_jogposition;
    MoveJ Align_4,v200,fine,tool_abs\WObj:=wobj0;
    err_write_jogposition;
    MoveJ Align_5,v200,fine,tool_abs\WObj:=wobj0;
    err_write_jogposition;
    MoveJ Align_6, v200, fine, tool_abs\WObj:=wobj0;
    err_write_jogposition;
    MoveJ Align_7, v200, fine, tool_abs\WObj:=wobj0;
    err_write_jogposition;
    MoveJ Align_8, v200, fine, tool_abs\WObj:=wobj0;
    err_write_jogposition;
    MoveJ Align_9, v200, fine, tool_abs\WObj:=wobj0;
    err_write_jogposition;
    MoveJ Align_10, v200, fine, tool_abs\WObj:=wobj0;
    err_write_jogposition;
    break;
  ENDPROC





  PROC new_calibration()
  number :=1;
    MoveJ calib_1,v200,fine,tool_abs\WObj:=wobj0;
    err_write_jogposition;
    MoveJ calib_2,v200,fine,tool_abs\WObj:=wobj0;
    err_write_jogposition;
    MoveJ calib_3,v200,fine,tool_abs\WObj:=wobj0;
    err_write_jogposition;
    MoveJ calib_4,v200,fine,tool_abs\WObj:=wobj0;
    err_write_jogposition;
    MoveJ calib_5,v200,fine,tool_abs\WObj:=wobj0;
    err_write_jogposition;
    MoveJ calib_6, v200, fine, tool_abs\WObj:=wobj0;
    err_write_jogposition;
    MoveJ calib_7, v200, fine, tool_abs\WObj:=wobj0;
    err_write_jogposition;
    MoveJ calib_8, v200, fine, tool_abs\WObj:=wobj0;
    err_write_jogposition;
    MoveJ calib_9, v200, fine, tool_abs\WObj:=wobj0;
    err_write_jogposition;
    MoveJ calib_10, v200, fine, tool_abs\WObj:=wobj0;
    err_write_jogposition;
    MoveJ calib_11,v200,fine,tool_abs\WObj:=wobj0;
    err_write_jogposition;
    MoveJ calib_12,v200,fine,tool_abs\WObj:=wobj0;
    err_write_jogposition;
    MoveJ calib_13,v200,fine,tool_abs\WObj:=wobj0;
    err_write_jogposition;
    MoveJ calib_14,v200,fine,tool_abs\WObj:=wobj0;
    err_write_jogposition;
    MoveJ calib_15,v200,fine,tool_abs\WObj:=wobj0;
    err_write_jogposition;
    MoveJ calib_16, v200, fine, tool_abs\WObj:=wobj0;
    err_write_jogposition;
    MoveJ calib_17, v200, fine, tool_abs\WObj:=wobj0;
    err_write_jogposition;
    MoveJ calib_18, v200, fine, tool_abs\WObj:=wobj0;
    err_write_jogposition;
    MoveJ calib_19, v200, fine, tool_abs\WObj:=wobj0;
    err_write_jogposition;
    MoveJ calib_20, v200, fine, tool_abs\WObj:=wobj0;
    err_write_jogposition;
    MoveJ calib_21,v200,fine,tool_abs\WObj:=wobj0;
    err_write_jogposition;
    MoveJ calib_22,v200,fine,tool_abs\WObj:=wobj0;
    err_write_jogposition;
    MoveJ calib_23,v200,fine,tool_abs\WObj:=wobj0;
    err_write_jogposition;
    MoveJ calib_24,v200,fine,tool_abs\WObj:=wobj0;
    err_write_jogposition;
    MoveJ calib_25,v200,fine,tool_abs\WObj:=wobj0;
    err_write_jogposition;
    MoveJ calib_26, v200, fine, tool_abs\WObj:=wobj0;
    err_write_jogposition;
    MoveJ calib_27, v200, fine, tool_abs\WObj:=wobj0;
    err_write_jogposition;
    MoveJ calib_28, v200, fine, tool_abs\WObj:=wobj0;
    err_write_jogposition;
    MoveJ calib_29, v200, fine, tool_abs\WObj:=wobj0;
    err_write_jogposition;
    MoveJ calib_30, v200, fine, tool_abs\WObj:=wobj0;
    err_write_jogposition;
    MoveJ calib_31,v200,fine,tool_abs\WObj:=wobj0;
    err_write_jogposition;
    MoveJ calib_32,v200,fine,tool_abs\WObj:=wobj0;
    err_write_jogposition;
    MoveJ calib_33,v200,fine,tool_abs\WObj:=wobj0;
    err_write_jogposition;
    MoveJ calib_34,v200,fine,tool_abs\WObj:=wobj0;
    err_write_jogposition;
    MoveJ calib_35,v200,fine,tool_abs\WObj:=wobj0;
    err_write_jogposition;
    MoveJ calib_36, v200, fine, tool_abs\WObj:=wobj0;
    err_write_jogposition;
    MoveJ calib_37, v200, fine, tool_abs\WObj:=wobj0;
    err_write_jogposition;
    MoveJ calib_38, v200, fine, tool_abs\WObj:=wobj0;
    err_write_jogposition;
    MoveJ calib_39, v200, fine, tool_abs\WObj:=wobj0;
    err_write_jogposition;
    MoveJ calib_40, v200, fine, tool_abs\WObj:=wobj0;
    err_write_jogposition;
    MoveJ calib_41,v200,fine,tool_abs\WObj:=wobj0;
    err_write_jogposition;
    MoveJ calib_42,v200,fine,tool_abs\WObj:=wobj0;
    err_write_jogposition;
    MoveJ calib_43,v200,fine,tool_abs\WObj:=wobj0;
    err_write_jogposition;
    MoveJ calib_44,v200,fine,tool_abs\WObj:=wobj0;
    err_write_jogposition;
    MoveJ calib_45,v200,fine,tool_abs\WObj:=wobj0;
    err_write_jogposition;
    MoveJ calib_46, v200, fine, tool_abs\WObj:=wobj0;
    err_write_jogposition;
    MoveJ calib_47, v200, fine, tool_abs\WObj:=wobj0;
    err_write_jogposition;
    MoveJ calib_48, v200, fine, tool_abs\WObj:=wobj0;
    err_write_jogposition;
    MoveJ calib_49, v200, fine, tool_abs\WObj:=wobj0;
    err_write_jogposition;
    MoveJ calib_50, v200, fine, tool_abs\WObj:=wobj0;
    err_write_jogposition;
    MoveJ calib_51,v200,fine,tool_abs\WObj:=wobj0;
    err_write_jogposition;
    MoveJ calib_52,v200,fine,tool_abs\WObj:=wobj0;
    err_write_jogposition;
    MoveJ calib_53,v200,fine,tool_abs\WObj:=wobj0;
    err_write_jogposition;
    MoveJ calib_54,v200,fine,tool_abs\WObj:=wobj0;
    err_write_jogposition;
    MoveJ calib_55,v200,fine,tool_abs\WObj:=wobj0;
    err_write_jogposition;
    MoveJ calib_56, v200, fine, tool_abs\WObj:=wobj0;
    err_write_jogposition;
    MoveJ calib_57, v200, fine, tool_abs\WObj:=wobj0;
    err_write_jogposition;
    MoveJ calib_58, v200, fine, tool_abs\WObj:=wobj0;
    err_write_jogposition;
    MoveJ calib_59, v200, fine, tool_abs\WObj:=wobj0;
    err_write_jogposition;
    MoveJ calib_60, v200, fine, tool_abs\WObj:=wobj0;
    err_write_jogposition;
    MoveJ calib_61,v200,fine,tool_abs\WObj:=wobj0;
    err_write_jogposition;
    MoveJ calib_62,v200,fine,tool_abs\WObj:=wobj0;
    err_write_jogposition;
    MoveJ calib_63,v200,fine,tool_abs\WObj:=wobj0;
    err_write_jogposition;
    MoveJ calib_64,v200,fine,tool_abs\WObj:=wobj0;
    err_write_jogposition;
    MoveJ calib_65,v200,fine,tool_abs\WObj:=wobj0;
    err_write_jogposition;
    MoveJ calib_66, v200, fine, tool_abs\WObj:=wobj0;
    err_write_jogposition;
    MoveJ calib_67, v200, fine, tool_abs\WObj:=wobj0;
    err_write_jogposition;
    MoveJ calib_68, v200, fine, tool_abs\WObj:=wobj0;
    err_write_jogposition;
    MoveJ calib_69, v200, fine, tool_abs\WObj:=wobj0;
    err_write_jogposition;
    MoveJ calib_70, v200, fine, tool_abs\WObj:=wobj0;
    err_write_jogposition;
    MoveJ calib_71,v200,fine,tool_abs\WObj:=wobj0;
    err_write_jogposition;
    MoveJ calib_72,v200,fine,tool_abs\WObj:=wobj0;
    err_write_jogposition;
    MoveJ calib_73,v200,fine,tool_abs\WObj:=wobj0;
    err_write_jogposition;
    MoveJ calib_74,v200,fine,tool_abs\WObj:=wobj0;
    err_write_jogposition;
    MoveJ calib_75,v200,fine,tool_abs\WObj:=wobj0;
    err_write_jogposition;
    MoveJ calib_76, v200, fine, tool_abs\WObj:=wobj0;
    err_write_jogposition;
    MoveJ calib_77, v200, fine, tool_abs\WObj:=wobj0;
    err_write_jogposition;
    MoveJ calib_78, v200, fine, tool_abs\WObj:=wobj0;
    err_write_jogposition;
    MoveJ calib_79, v200, fine, tool_abs\WObj:=wobj0;
    err_write_jogposition;
    MoveJ calib_80, v200, fine, tool_abs\WObj:=wobj0;
    err_write_jogposition;
    MoveJ calib_81,v200,fine,tool_abs\WObj:=wobj0;
    err_write_jogposition;
    MoveJ calib_82,v200,fine,tool_abs\WObj:=wobj0;
    err_write_jogposition;
    MoveJ calib_83,v200,fine,tool_abs\WObj:=wobj0;
    err_write_jogposition;
    MoveJ calib_84,v200,fine,tool_abs\WObj:=wobj0;
    err_write_jogposition;
    MoveJ calib_85,v200,fine,tool_abs\WObj:=wobj0;
    err_write_jogposition;
    MoveJ calib_86, v200, fine, tool_abs\WObj:=wobj0;
    err_write_jogposition;
    MoveJ calib_87, v200, fine, tool_abs\WObj:=wobj0;
    err_write_jogposition;
    MoveJ calib_88, v200, fine, tool_abs\WObj:=wobj0;
    err_write_jogposition;
    MoveJ calib_89, v200, fine, tool_abs\WObj:=wobj0;
    err_write_jogposition;
    MoveJ calib_90, v200, fine, tool_abs\WObj:=wobj0;
    err_write_jogposition;
    MoveJ calib_91,v200,fine,tool_abs\WObj:=wobj0;
    err_write_jogposition;
    MoveJ calib_92,v200,fine,tool_abs\WObj:=wobj0;
    err_write_jogposition;
    MoveJ calib_93,v200,fine,tool_abs\WObj:=wobj0;
    err_write_jogposition;
    MoveJ calib_94,v200,fine,tool_abs\WObj:=wobj0;
    err_write_jogposition;
    MoveJ calib_95,v200,fine,tool_abs\WObj:=wobj0;
    err_write_jogposition;
    MoveJ calib_96, v200, fine, tool_abs\WObj:=wobj0;
    err_write_jogposition;
    MoveJ calib_97, v200, fine, tool_abs\WObj:=wobj0;
    err_write_jogposition;
    MoveJ calib_98, v200, fine, tool_abs\WObj:=wobj0;
    err_write_jogposition;
    MoveJ calib_99, v200, fine, tool_abs\WObj:=wobj0;
    err_write_jogposition;
    MoveJ calib_100, v200, fine, tool_abs\WObj:=wobj0;
    err_write_jogposition;
    break;


  ENDPROC

 PROC TcpVerify1()
    MoveL [[1384,593,915],[0.632261,-0.365612,0.594547,-0.336285],[0,0,2,1],[0,9E+09,9E+09,0.00772622,0.0471901,0.00028478]], v1000, z50, tool0;
    MoveL [[884,593,915],[0.632261,-0.365612,0.594547,-0.336285],[0,0,2,1],[0,9E+09,9E+09,0.00772622,0.0471901,0.00028478]], v1000, z50, tool0;
    MoveL [[1384,93,915],[0.632261,-0.365612,0.594547,-0.336285],[0,0,2,1],[0,9E+09,9E+09,0.00772622,0.0471901,0.00028478]], v1000, z50, tool0;
    MoveL [[1384,593,1415],[0.632261,-0.365612,0.594547,-0.336285],[0,0,2,1],[0,9E+09,9E+09,0.00772622,0.0471901,0.00028478]], v1000, z50, tool0;




 ENDPROC

 PROC TcpVerify2()
    MoveL [[1625,-669,583],[0.667372,-0.403997,0.554082,-0.290507],[-1,-1,3,1],[0,9E+09,9E+09,0.00858047,0.0845895,0.000234465]], v1000, z50, tool0;
    MoveL [[1125,-669,583],[0.667372,-0.403997,0.554082,-0.290507],[-1,-1,3,1],[0,9E+09,9E+09,0.00858047,0.0845895,0.000234465]], v1000, z50, tool0;
    MoveL [[1625,-169,583],[0.667372,-0.403997,0.554082,-0.290507],[-1,-1,3,1],[0,9E+09,9E+09,0.00858047,0.0845895,0.000234465]], v1000, z50, tool0;
    MoveL [[1625,-669,83],[0.667372,-0.403997,0.554082,-0.290507],[-1,-1,3,1],[0,9E+09,9E+09,0.00858047,0.0845895,0.000234465]], v1000, z50, tool0;




 ENDPROC

 PROC TcpVerify3()
     number :=1;
     ErrWrite \w,"test","ABSACC";
     ErrWrite \w,"ready??????","ABSACC";

	    MoveAbsJ JT_Set1_1,v200,fine,tool_abs\WObj:=wobj0;
         current_pos := CRobT(\Tool:=tool_abs \WObj:=wobj0);
         log_string := "X:" + NumToStr(current_pos.trans.x, 2) + ", " +
                     "Y:" + NumToStr(current_pos.trans.y, 2) + ", " +
                     "Z:" + NumToStr(current_pos.trans.z, 2) + ", " +
                     "Q1:" + NumToStr(current_pos.rot.q1, 4) + ", " +
                     "Q2:" + NumToStr(current_pos.rot.q2, 4) + ", " +
                     "Q3:" + NumToStr(current_pos.rot.q3, 4) + ", " +
                     "Q4:" + NumToStr(current_pos.rot.q4, 4);

        ErrWrite \w,log_string,"ABSACC";
        err_write_position;
        MoveL [[431,-90,1782],[0.689633,-0.0852204,0.712187,0.0996667],[-1,0,-1,0],[0,9E+09,9E+09,0.00958726,0.0242127,0.000143899]], v1000, z50, tool0;
        MoveL [[931,-590,1782],[0.689633,-0.0852204,0.712187,0.0996667],[-1,0,-1,0],[0,9E+09,9E+09,0.00958726,0.0242127,0.000143899]], v1000, z50, tool0;
        MoveL [[931,-90,1282],[0.689633,-0.0852204,0.712187,0.0996667],[-1,0,-1,0],[0,9E+09,9E+09,0.00958726,0.0242127,0.000143899]], v1000, z50, tool0;

 ENDPROC


  PROC Calibration()
    number :=1;
	MoveAbsJ JT_Set1_1,v200,fine,tool_abs\WObj:=wobj0;
    err_write_position;
    MoveAbsJ JT_Set1_2,v200,fine,tool_abs\WObj:=wobj0;
    err_write_position;
    MoveAbsJ JT_Set1_3,v200,fine,tool_abs\WObj:=wobj0;
    err_write_position;
    MoveAbsJ JT_Set1_4,v200,fine,tool_abs\WObj:=wobj0;
    err_write_position;
    MoveAbsJ JT_Set1_5,v200,fine,tool_abs\WObj:=wobj0;
    err_write_position;
    MoveAbsJ JT_Set1_6,v200,fine,tool_abs\WObj:=wobj0;err_write_position;
    MoveAbsJ JT_Set1_7,v200,fine,tool_abs\WObj:=wobj0;err_write_position;
    MoveAbsJ JT_Set1_8,v200,fine,tool_abs\WObj:=wobj0;err_write_position;
    MoveAbsJ JT_Set1_9,v200,fine,tool_abs\WObj:=wobj0;err_write_position;
    MoveAbsJ JT_Set1_10,v200,fine,tool_abs\WObj:=wobj0;err_write_position;
    MoveAbsJ JT_Set1_11,v200,fine,tool_abs\WObj:=wobj0;err_write_position;
    MoveAbsJ JT_Set1_12,v200,fine,tool_abs\WObj:=wobj0;err_write_position;
    MoveAbsJ JT_Set1_13,v200,fine,tool_abs\WObj:=wobj0;err_write_position;
    MoveAbsJ JT_Set1_14,v200,fine,tool_abs\WObj:=wobj0;err_write_position;
    MoveAbsJ JT_Set1_15,v200,fine,tool_abs\WObj:=wobj0;err_write_position;
    MoveAbsJ JT_Set1_16,v200,fine,tool_abs\WObj:=wobj0;err_write_position;
    MoveAbsJ JT_Set1_17,v200,fine,tool_abs\WObj:=wobj0;err_write_position;
    MoveAbsJ JT_Set1_18,v200,fine,tool_abs\WObj:=wobj0;err_write_position;
    MoveAbsJ JT_Set1_19,v200,fine,tool_abs\WObj:=wobj0;err_write_position;
    MoveAbsJ JT_Set1_20,v200,fine,tool_abs\WObj:=wobj0;err_write_position;
    MoveAbsJ JT_Set1_21,v200,fine,tool_abs\WObj:=wobj0;err_write_position;
    MoveAbsJ JT_Set1_22,v200,fine,tool_abs\WObj:=wobj0;err_write_position;
    MoveAbsJ JT_Set1_23,v200,fine,tool_abs\WObj:=wobj0;err_write_position;
    MoveAbsJ JT_Set1_24,v200,fine,tool_abs\WObj:=wobj0;err_write_position;
    MoveAbsJ JT_Set1_25,v200,fine,tool_abs\WObj:=wobj0;err_write_position;
    MoveAbsJ JT_Set1_26,v200,fine,tool_abs\WObj:=wobj0;err_write_position;
    MoveAbsJ JT_Set1_27,v200,fine,tool_abs\WObj:=wobj0;err_write_position;
    MoveAbsJ JT_Set1_28,v200,fine,tool_abs\WObj:=wobj0;err_write_position;
    MoveAbsJ JT_Set1_29,v200,fine,tool_abs\WObj:=wobj0;err_write_position;
    MoveAbsJ JT_Set1_30,v200,fine,tool_abs\WObj:=wobj0;err_write_position;
    MoveAbsJ JT_Set1_31,v200,fine,tool_abs\WObj:=wobj0;err_write_position;
    MoveAbsJ JT_Set1_32,v200,fine,tool_abs\WObj:=wobj0;err_write_position;
    MoveAbsJ JT_Set1_33,v200,fine,tool_abs\WObj:=wobj0;err_write_position;
    MoveAbsJ JT_Set1_34,v200,fine,tool_abs\WObj:=wobj0;err_write_position;
    MoveAbsJ JT_Set1_35,v200,fine,tool_abs\WObj:=wobj0;err_write_position;
    MoveAbsJ JT_Set1_36,v200,fine,tool_abs\WObj:=wobj0;err_write_position;
    MoveAbsJ JT_Set1_37,v200,fine,tool_abs\WObj:=wobj0;err_write_position;
    MoveAbsJ JT_Set1_38,v200,fine,tool_abs\WObj:=wobj0;err_write_position;
    MoveAbsJ JT_Set1_39,v200,fine,tool_abs\WObj:=wobj0;err_write_position;
    MoveAbsJ JT_Set1_40,v200,fine,tool_abs\WObj:=wobj0;err_write_position;
    MoveAbsJ JT_Set1_41,v200,fine,tool_abs\WObj:=wobj0;err_write_position;
    MoveAbsJ JT_Set1_42,v200,fine,tool_abs\WObj:=wobj0;err_write_position;
    MoveAbsJ JT_Set1_43,v200,fine,tool_abs\WObj:=wobj0;err_write_position;
    MoveAbsJ JT_Set1_44,v200,fine,tool_abs\WObj:=wobj0;err_write_position;
    MoveAbsJ JT_Set1_45,v200,fine,tool_abs\WObj:=wobj0;err_write_position;
    MoveAbsJ JT_Set1_46,v200,fine,tool_abs\WObj:=wobj0;err_write_position;
    MoveAbsJ JT_Set1_47,v200,fine,tool_abs\WObj:=wobj0;err_write_position;
    MoveAbsJ JT_Set1_48,v200,fine,tool_abs\WObj:=wobj0;err_write_position;
    MoveAbsJ JT_Set1_49,v200,fine,tool_abs\WObj:=wobj0;err_write_position;
    MoveAbsJ JT_Set1_50,v200,fine,tool_abs\WObj:=wobj0;err_write_position;
    MoveAbsJ JT_Set1_51,v200,fine,tool_abs\WObj:=wobj0;err_write_position;
    MoveAbsJ JT_Set1_52,v200,fine,tool_abs\WObj:=wobj0;err_write_position;
    MoveAbsJ JT_Set1_53,v200,fine,tool_abs\WObj:=wobj0;err_write_position;
    MoveAbsJ JT_Set1_54,v200,fine,tool_abs\WObj:=wobj0;err_write_position;
    MoveAbsJ JT_Set1_55,v200,fine,tool_abs\WObj:=wobj0;err_write_position;
    MoveAbsJ JT_Set1_56,v200,fine,tool_abs\WObj:=wobj0;err_write_position;
    MoveAbsJ JT_Set1_57,v200,fine,tool_abs\WObj:=wobj0;err_write_position;
    MoveAbsJ JT_Set1_58,v200,fine,tool_abs\WObj:=wobj0;err_write_position;
    MoveAbsJ JT_Set1_59,v200,fine,tool_abs\WObj:=wobj0;err_write_position;
    MoveAbsJ JT_Set1_60,v200,fine,tool_abs\WObj:=wobj0;err_write_position;
    MoveAbsJ JT_Set1_61,v200,fine,tool_abs\WObj:=wobj0;err_write_position;
    MoveAbsJ JT_Set1_62,v200,fine,tool_abs\WObj:=wobj0;err_write_position;
    MoveAbsJ JT_Set1_63,v200,fine,tool_abs\WObj:=wobj0;err_write_position;
    MoveAbsJ JT_Set1_64,v200,fine,tool_abs\WObj:=wobj0;err_write_position;
    MoveAbsJ JT_Set1_65,v200,fine,tool_abs\WObj:=wobj0;err_write_position;
    MoveAbsJ JT_Set1_66,v200,fine,tool_abs\WObj:=wobj0;err_write_position;
    MoveAbsJ JT_Set1_67,v200,fine,tool_abs\WObj:=wobj0;err_write_position;
    MoveAbsJ JT_Set1_68,v200,fine,tool_abs\WObj:=wobj0;err_write_position;
    MoveAbsJ JT_Set1_69,v200,fine,tool_abs\WObj:=wobj0;err_write_position;
    MoveAbsJ JT_Set1_70,v200,fine,tool_abs\WObj:=wobj0;err_write_position;
    MoveAbsJ JT_Set1_71,v200,fine,tool_abs\WObj:=wobj0;err_write_position;
    MoveAbsJ JT_Set1_72,v200,fine,tool_abs\WObj:=wobj0;err_write_position;
    MoveAbsJ JT_Set1_73,v200,fine,tool_abs\WObj:=wobj0;err_write_position;
    MoveAbsJ JT_Set1_74,v200,fine,tool_abs\WObj:=wobj0;err_write_position;
    MoveAbsJ JT_Set1_75,v200,fine,tool_abs\WObj:=wobj0;err_write_position;
    MoveAbsJ JT_Set1_76,v200,fine,tool_abs\WObj:=wobj0;err_write_position;
    MoveAbsJ JT_Set1_77,v200,fine,tool_abs\WObj:=wobj0;err_write_position;
    MoveAbsJ JT_Set1_78,v200,fine,tool_abs\WObj:=wobj0;err_write_position;
    MoveAbsJ JT_Set1_79,v200,fine,tool_abs\WObj:=wobj0;err_write_position;
    MoveAbsJ JT_Set1_80,v200,fine,tool_abs\WObj:=wobj0;err_write_position;
    MoveAbsJ JT_Set1_81,v200,fine,tool_abs\WObj:=wobj0;err_write_position;
    MoveAbsJ JT_Set1_82,v200,fine,tool_abs\WObj:=wobj0;err_write_position;
    MoveAbsJ JT_Set1_83,v200,fine,tool_abs\WObj:=wobj0;err_write_position;
    MoveAbsJ JT_Set1_84,v200,fine,tool_abs\WObj:=wobj0;err_write_position;
    MoveAbsJ JT_Set1_85,v200,fine,tool_abs\WObj:=wobj0;err_write_position;
    MoveAbsJ JT_Set1_86,v200,fine,tool_abs\WObj:=wobj0;err_write_position;
    MoveAbsJ JT_Set1_87,v200,fine,tool_abs\WObj:=wobj0;err_write_position;
    MoveAbsJ JT_Set1_88,v200,fine,tool_abs\WObj:=wobj0;err_write_position;
    MoveAbsJ JT_Set1_89,v200,fine,tool_abs\WObj:=wobj0;err_write_position;
    MoveAbsJ JT_Set1_90,v200,fine,tool_abs\WObj:=wobj0;err_write_position;
    MoveAbsJ JT_Set1_91,v200,fine,tool_abs\WObj:=wobj0;err_write_position;
    MoveAbsJ JT_Set1_92,v200,fine,tool_abs\WObj:=wobj0;err_write_position;
    MoveAbsJ JT_Set1_93,v200,fine,tool_abs\WObj:=wobj0;err_write_position;
    MoveAbsJ JT_Set1_94,v200,fine,tool_abs\WObj:=wobj0;err_write_position;
    MoveAbsJ JT_Set1_95,v200,fine,tool_abs\WObj:=wobj0;err_write_position;
    MoveAbsJ JT_Set1_96,v200,fine,tool_abs\WObj:=wobj0;err_write_position;
    MoveAbsJ JT_Set1_97,v200,fine,tool_abs\WObj:=wobj0;err_write_position;
    MoveAbsJ JT_Set1_98,v200,fine,tool_abs\WObj:=wobj0;err_write_position;
    MoveAbsJ JT_Set1_99,v200,fine,tool_abs\WObj:=wobj0;err_write_position;
    MoveAbsJ JT_Set1_100,v200,fine,tool_abs\WObj:=wobj0;err_write_position;
  ENDPROC





 PROC CalibAxis7()
	MoveJ CalibAxis7_1, v1500, fine, tool_abs\WObj:=wobj0;
    MoveJ CalibAxis7_2,v200,fine,tool_abs\WObj:=wobj0;
    MoveJ CalibAxis7_3,v200,fine,tool_abs\WObj:=wobj0;
    MoveJ CalibAxis7_4,v200,fine,tool_abs\WObj:=wobj0;
    MoveJ CalibAxis7_5,v200,fine,tool_abs\WObj:=wobj0;
    MoveJ CalibAxis7_6, v200, fine, tool_abs\WObj:=wobj0;
    MoveJ CalibAxis7_7, v200, fine, tool_abs\WObj:=wobj0;
    MoveJ CalibAxis7_8, v200, fine, tool_abs\WObj:=wobj0;
    MoveJ CalibAxis7_9, v200, fine, tool_abs\WObj:=wobj0;
    MoveJ CalibAxis7_10, v200, fine, tool_abs\WObj:=wobj0;
    MoveJ CalibAxis7_11,v200,fine,tool_abs\WObj:=wobj0;
    MoveJ CalibAxis7_12,v200,fine,tool_abs\WObj:=wobj0;
    MoveJ CalibAxis7_13,v200,fine,tool_abs\WObj:=wobj0;
    MoveJ CalibAxis7_14,v200,fine,tool_abs\WObj:=wobj0;
    MoveJ CalibAxis7_15,v200,fine,tool_abs\WObj:=wobj0;
    MoveJ CalibAxis7_16, v200, fine, tool_abs\WObj:=wobj0;
    MoveJ CalibAxis7_17, v200, fine, tool_abs\WObj:=wobj0;
    MoveJ CalibAxis7_18, v200, fine, tool_abs\WObj:=wobj0;
    MoveJ CalibAxis7_19, v200, fine, tool_abs\WObj:=wobj0;
    MoveJ CalibAxis7_20, v200, fine, tool_abs\WObj:=wobj0;
 ENDPROC


 PROC CalibAxis8()
	MoveJ CalibAxis8_1, v1500, fine, tool_abs\WObj:=wobj0;
    MoveJ CalibAxis8_2,v200,fine,tool_abs\WObj:=wobj0;
    MoveJ CalibAxis8_3,v200,fine,tool_abs\WObj:=wobj0;
    MoveJ CalibAxis8_4,v200,fine,tool_abs\WObj:=wobj0;
    MoveJ CalibAxis8_5,v200,fine,tool_abs\WObj:=wobj0;
    MoveJ CalibAxis8_6, v200, fine, tool_abs\WObj:=wobj0;
    MoveJ CalibAxis8_7, v200, fine, tool_abs\WObj:=wobj0;
    MoveJ CalibAxis8_8, v200, fine, tool_abs\WObj:=wobj0;
    MoveJ CalibAxis8_9, v200, fine, tool_abs\WObj:=wobj0;
    MoveJ CalibAxis8_10, v200, fine, tool_abs\WObj:=wobj0;
    MoveJ CalibAxis8_11,v200,fine,tool_abs\WObj:=wobj0;
    MoveJ CalibAxis8_12,v200,fine,tool_abs\WObj:=wobj0;
    MoveJ CalibAxis8_13,v200,fine,tool_abs\WObj:=wobj0;
    MoveJ CalibAxis8_14,v200,fine,tool_abs\WObj:=wobj0;
    MoveJ CalibAxis8_15,v200,fine,tool_abs\WObj:=wobj0;
    MoveJ CalibAxis8_16, v200, fine, tool_abs\WObj:=wobj0;
    MoveJ CalibAxis8_17, v200, fine, tool_abs\WObj:=wobj0;
    MoveJ CalibAxis8_18, v200, fine, tool_abs\WObj:=wobj0;
    MoveJ CalibAxis8_19, v200, fine, tool_abs\WObj:=wobj0;
    MoveJ CalibAxis8_20, v200, fine, tool_abs\WObj:=wobj0;
 ENDPROC

 PROC CalibAxis9()

 ENDPROC


 PROC Calibration_move_to_home()
    !ActUnit STN1;
    number :=0;
	MoveAbsJ [[0,0,0,0,0,0],[0,9E+09,9E+09,0,0,0]],v200,fine,tool_abs\WObj:=wobj0;
    err_write_position;
    !DeactUnit STN1;
 ENDPROC

 PROC err_write_jogposition()
    WaitRob\InPos;
    currentjoints :=CJointT();
    rob_axis_1 :=currentjoints.robax.rax_1;
    rob_axis_2 :=currentjoints.robax.rax_2;
    rob_axis_3 :=currentjoints.robax.rax_3;
    rob_axis_4 :=currentjoints.robax.rax_4;
    rob_axis_5 :=currentjoints.robax.rax_5;
    rob_axis_6 :=currentjoints.robax.rax_6;
     log_string := "P:"+outnumber+"," + NumToStr(currentjoints.robax.rax_1, 5)  +
                     "," + NumToStr(currentjoints.robax.rax_2, 5) +
                     "," + NumToStr(currentjoints.robax.rax_3, 5) +
                     "," + NumToStr(currentjoints.robax.rax_4, 3)  +
                     "," + NumToStr(currentjoints.robax.rax_5, 3) +
                     "," + NumToStr(currentjoints.robax.rax_6, 3) ;
    ErrWrite \w,log_string,"ABSACC";
    TPWrite log_string;
 ENDPROC

PROC err_write_position()
    WaitRob\InPos;
    current_pos := CRobT(\Tool:=tool_abs \WObj:=wobj0);
outnumber :=NumToStr(number,0);

    number := number +1;
log_string := "P:"+outnumber+"," + NumToStr(current_pos.trans.x, 2)  +
                     "," + NumToStr(current_pos.trans.y, 2) +
                     "," + NumToStr(current_pos.trans.z, 2) +
                     "," + NumToStr(current_pos.rot.q1, 2)  +
                     "," + NumToStr(current_pos.rot.q2, 2) +
                     "," + NumToStr(current_pos.rot.q3, 2) +
                     "," + NumToStr(current_pos.rot.q4, 2);
     ErrWrite \w,log_string,"ABSACC";
     TPWrite log_string;


    jt_current :=CJointT();

    rt_current :=CalcRobT(jt_current,tool_abs \WObj:=wobj0);
    x_pos := rt_current.trans.x;
    y_pos := rt_current.trans.y;
    z_pos := rt_current.trans.z;
    q1_pos := rt_current.rot.q1;
    q2_pos :=rt_current.rot.q2;
    q3_pos :=rt_current.rot.q3;
    q4_pos :=rt_current.rot.q4;
    TPWrite "x"\num:=x_pos;
    TPWrite "y"\num:=y_pos;
    TPWrite "z"\num:=z_pos;
    log_string := "P:"+outnumber+"," + NumToStr(current_pos.trans.x, 5)  +
                     "," + NumToStr(current_pos.trans.y, 5) +
                     "," + NumToStr(current_pos.trans.z, 5) +
                     "," + NumToStr(current_pos.rot.q1, 3)  +
                     "," + NumToStr(current_pos.rot.q2, 3) +
                     "," + NumToStr(current_pos.rot.q3, 3) +
                     "," + NumToStr(current_pos.rot.q4, 3);
    ErrWrite \w,log_string,"ABSACC";
    TPWrite log_string;


     break;
ENDPROC

  PROC RecordPosition_abs()

        current_pos := CRobT(\Tool:=tool_abs \WObj:=wobj0);


        log_string := "X:" + NumToStr(current_pos.trans.x, 2) + ", " +
                     "Y:" + NumToStr(current_pos.trans.y, 2) + ", " +
                     "Z:" + NumToStr(current_pos.trans.z, 2) + ", " +
                     "Q1:" + NumToStr(current_pos.rot.q1, 4) + ", " +
                     "Q2:" + NumToStr(current_pos.rot.q2, 4) + ", " +
                     "Q3:" + NumToStr(current_pos.rot.q3, 4) + ", " +
                     "Q4:" + NumToStr(current_pos.rot.q4, 4);

        ! ????
        Write file_no, log_string;
        ErrWrite \w,"screen!!!!!!!!!!!!!!!!!!!!!!!!!!!!!!","ABSACC";
    ENDPROC


ENDMODULE
